(* Logix 5000 project; controller AdvManLab vendor 1 type 14 code 158 rev 28.12; software revision 28.01; part 13 of 13 *)
(* tags used below, declared in another part *)
   Auto_Valves_Safe01 : SINT;
   Auto_Valves_Safe02 : SINT;
   Man_Valves_Safe01 : SINT;
   Man_Valves_Safe02 : SINT;
   Mode_Auto_Safe : BOOL;
   Mode_Manual_Safe : BOOL;
   Mode_None_Safe : BOOL;
   ValvesOff : SINT;
(* SafetyProgram, continued *)

ROUTINE ValveManifold   (* ladder *)
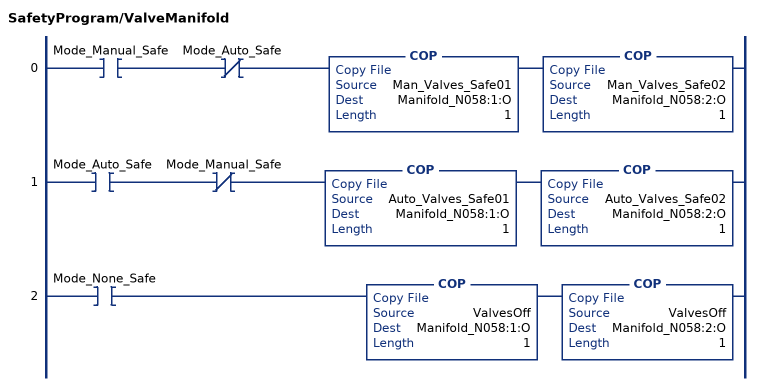
   0: XIC(Mode_Manual_Safe)XIO(Mode_Auto_Safe)COP(Man_Valves_Safe01,Manifold_N058:1:O,1)COP(Man_Valves_Safe02,Manifold_N058:2:O,1);
   1: XIC(Mode_Auto_Safe)XIO(Mode_Manual_Safe)COP(Auto_Valves_Safe01,Manifold_N058:1:O,1)COP(Auto_Valves_Safe02,Manifold_N058:2:O,1);
   2: XIC(Mode_None_Safe)COP(ValvesOff,Manifold_N058:1:O,1)COP(ValvesOff,Manifold_N058:2:O,1);
END_ROUTINE
END_PROGRAM
